{attribute 'qualified_only'}
{attribute 'strict'}
{attribute 'to_string'}
TYPE TestFlexiBufferState :
(
	INIT,
	ADD_ELEMENT,
	REMOVE_ELEMENT,
	WAIT
);
END_TYPE

(* stored: Version 1.1.0.1
   DUT TestFlexiBufferState: Id {0a35cf6a-30e8-4a67-8f12-0005a74732e3} *)
